INTERFACE ITF_TopElement EXTENDS ITF_BaseTopElement

END_INTERFACE

(* stored: Version 1.1.0.1, ProductVersion 3.1.4024.15
   Itf ITF_TopElement: Id {f946a41b-c75b-42d1-a052-4384bb0e99a9} *)
